# B&R Automation Studio project simulation_of_controlling_the_barn_door
Automation Studio 4.2.10.53 SP

## Configuration SampleText

CPU 4PP065.0571-P74, AutomationRuntime D4.26, Build 4.1.2, Vc V4.25.0, Safety 1.6

### Task classes (Cpu.sw)
```
Cyclic#1 (cycle 2000 us, tolerance 0 us):
  ncsdcctrl <- ncsdcctrl.prg
Cyclic#4 (cycle 100000 us, tolerance 100000 us):
  Program <- Program.prg
NcDataObjects: acp10etxen <- acp10etxen.dob, gAxis01a <- gAxis01obj.gAxis01a.dob, gAxis01i <- gAxis01obj.gAxis01i.dob
Libraries: Acp10sdc, sys_lib, Runtime, asstring, Acp10man, Acp10par, NcGlobal, Acp10_MC, brsystem, AsBrStr, Library
```

### Hardware
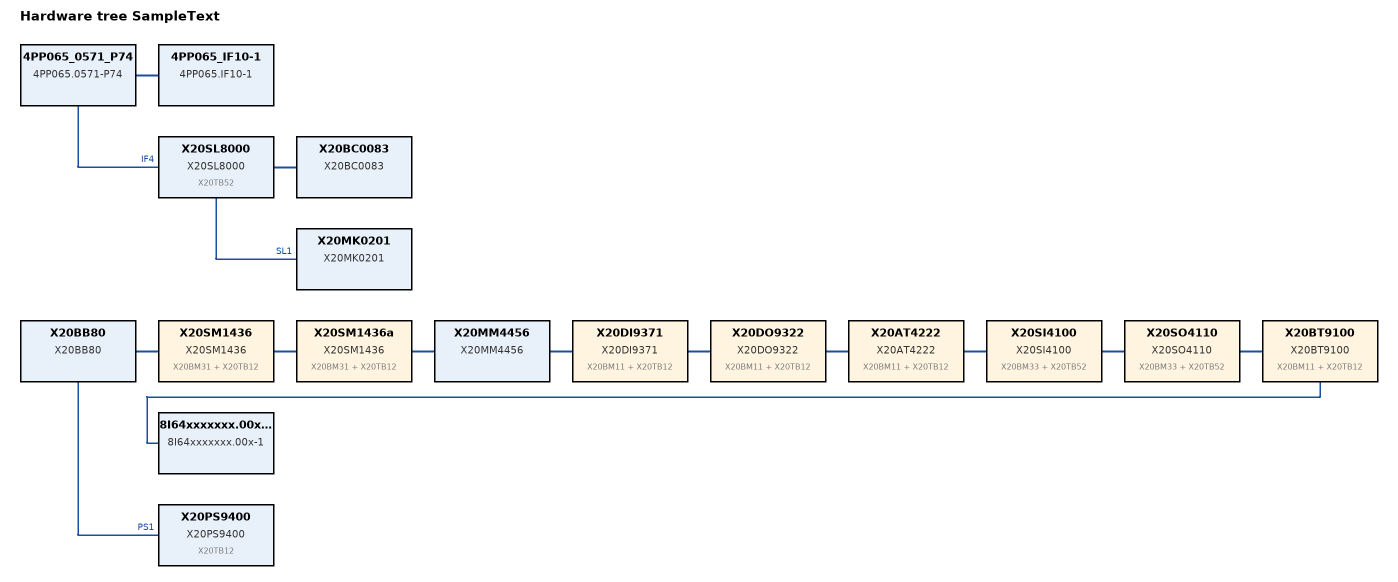
```
4PP065_0571_P74 : 4PP065.0571-P74 v1.1.1.0
  Connector IF4:
    EplInterfaceRedundant = 0
    EplEthInterfaceRedundant = 0
  Connector IF5:
    ActivateDevice = 1
    Mode = Manual
    InternetAddress = 10.1.1.13
    SubnetMask = 255.255.255.0
  ConfigurationID = DriveControl_SampleText
  TimerDeviceType = EPLX2X
  TimerDevice = 4PP065_0571_P74.IF4
  TaskClassIdleTime = 2000
  Cyclic1Duration = 2000
  Cyclic1Tolerance = 0
  Cyclic1Output = 1
  Cyclic2Duration = 20000
  Cyclic2Tolerance = 20000
  Cyclic3Duration = 50000
  Cyclic3Tolerance = 50000
  Cyclic4Duration = 100000
  Cyclic4Tolerance = 100000
  Cyclic5Duration = 200000
  Cyclic5Tolerance = 200000
  Cyclic6Duration = 500000
  Cyclic6Tolerance = 500000
  Cyclic7Duration = 1000000
  Cyclic7Tolerance = 1000000
  Cyclic8Duration = 10000
  Cyclic8Tolerance = 30000000
4PP065_IF10-1 : 4PP065.IF10-1 v1.0.2.0  [SS -> 4PP065_0571_P74.SS1]
8I64xxxxxxx.00x-1 : 8I64xxxxxxx.00x-1 v1.3.8.5  [X2X1 -> X20BT9100.X2X1]
  packedETAD = packed
  packedETI = packed
  packedCMDD = packed
  packedCMI = packed
  ACC = 30
X20AT4222 : X20AT4222 v1.2.1.0  [SS1 -> X20TB12e.SS; SL -> X20BM11c.SL1]
X20BB80 : X20BB80 v1.0.0.2
X20BC0083 : X20BC0083 v2.5.0.0  [PLK1 -> X20SL8000.PLK2 (NodeNumber=2); SL -> X20BB80.SL1]
X20BM11 : X20BM11 v1.0.0.1  [X2X1 -> X20BM33a.X2X2]
X20BM11a : X20BM11 v1.0.0.1  [X2X1 -> X20MM4456.X2X2]
X20BM11b : X20BM11 v1.0.0.1  [X2X1 -> X20BM11a.X2X2]
X20BM11c : X20BM11 v1.0.0.1  [X2X1 -> X20BM11b.X2X2]
X20BM31 : X20BM31 v1.0.0.1  [X2X1 -> X20BB80.IF1]
X20BM31a : X20BM31 v1.0.0.1  [X2X1 -> X20BM31.X2X2]
X20BM33 : X20BM33 v1.0.0.4  [X2X1 -> X20BM11c.X2X2]
X20BM33a : X20BM33 v1.0.0.4  [X2X1 -> X20BM33.X2X2]
X20BT9100 : X20BT9100 v1.0.2.4  [SS1 -> X20TB12f.SS; SL -> X20BM11.SL1]
X20DI9371 : X20DI9371 v1.0.1.3  [SS1 -> X20TB12c.SS; SL -> X20BM11a.SL1]
X20DO9322 : X20DO9322 v1.0.3.0  [SS1 -> X20TB12d.SS; SL -> X20BM11b.SL1]
X20MK0201 : X20MK0201 v1.0.0.0  [SL -> X20SL8000.SL1]
X20MM4456 : X20MM4456 v1.1.3.1  [X2X1 -> X20BM31a.X2X2]
X20PS9400 : X20PS9400 v1.0.2.4  [SS1 -> X20TB12.SS; PS -> X20BB80.PS1]
X20SI4100 : X20SI4100 v1.10.0.1  [SS1 -> X20TB52.SS; SL -> X20BM33.SL1]
X20SL8000 : X20SL8000 v1.6.5.1  [PLK1 -> 4PP065_0571_P74.IF4 (NodeNumber=1); PLK2 -> X20BC0083.PLK1 (NodeNumber=1); SS1 -> X20TB52b.SS]
  SafeProject = SafeLOGIC-1
X20SM1436 : X20SM1436 v1.4.2.0  [SS1 -> X20TB12a.SS; SL -> X20BM31.SL1]
X20SM1436a : X20SM1436 v1.4.2.0  [SS1 -> X20TB12b.SS; SL -> X20BM31a.SL1]
X20SO4110 : X20SO4110 v1.10.0.1  [SS1 -> X20TB52a.SS; SL -> X20BM33a.SL1]
  SafeModuleID = 3
X20TB12 : X20TB12 v1.0.0.0
X20TB12a : X20TB12 v1.0.0.0
X20TB12b : X20TB12 v1.0.0.0
X20TB12c : X20TB12 v1.0.0.0
X20TB12d : X20TB12 v1.0.0.0
X20TB12e : X20TB12 v1.0.0.0
X20TB12f : X20TB12 v1.0.0.0
X20TB52 : X20TB52 v1.0.0.1
X20TB52a : X20TB52 v1.0.0.1
X20TB52b : X20TB52 v1.0.0.1
```

### IoMap.iom - 4PP065_0571_P74/IoMap.iom
```iecst
VAR_CONFIG
	Cyclic#1.gAxis01_DrvIf.iLifeCnt AT %IB."8I64xxxxxxx.00x-1".SDC_LifeCnt;
	Cyclic#1.gAxis01_DrvIf.oSetTime AT %QW."8I64xxxxxxx.00x-1".SDC_SetTime;
	Cyclic#1.gAxis01_DrvIf.oSetPos AT %QW."8I64xxxxxxx.00x-1".LFRD_Output;
	Cyclic#1.gAxis01_DiDoIf.iLifeCntDriveReady AT %IB."8I64xxxxxxx.00x-1".SDC_LifeCnt;
	Cyclic#1.gAxis01_DiDoIf.iLifeCntDriveEnable AT %IB."8I64xxxxxxx.00x-1".SDC_LifeCnt;
	Cyclic#1.gAxis01_ModuleOk AT %IX."8I64xxxxxxx.00x-1".ModuleOk;
	::Program:FBDoorSM.direction AT %IX."X20DI9371".DigitalInput01;
	::Program:FBDoorSM.sw1 AT %IX."X20DI9371".DigitalInput02;
	::Program:FBDoorSM.sw2 AT %IX."X20DI9371".DigitalInput03;
	::Program:FBDoorSM.sw3 AT %IX."X20DI9371".DigitalInput04;
	::Program:FBDoorSM.sw4 AT %IX."X20DI9371".DigitalInput05;
	::Program:FBLedSM.led1 AT %QX."X20DO9322".DigitalOutput01;
	::Program:FBLedSM.led2 AT %QX."X20DO9322".DigitalOutput02;
	::Program:FBLedSM.led3 AT %QX."X20DO9322".DigitalOutput03;
	::Program:FBLedSM.led4 AT %QX."X20DO9322".DigitalOutput04;
	::Program:FBDriveSM.state AT %IW."8I64xxxxxxx.00x-1".ETAD_Input;
	::Program:FBDriveSM.command AT %IW."8I64xxxxxxx.00x-1".ETI_Input;
	::Program:FBDriveSM.speed AT %IW."8I64xxxxxxx.00x-1".RFRD_Input;
END_VAR
```

## Logical view

Binary libraries used (declarations not repeated): Runtime, Operator, AsIecCon, astime, sys_lib, asstring, Acp10sdc 3.16.2, Acp10man 3.16.2, Acp10par 3.16.2, NcGlobal 3.16.2, Acp10_MC 3.16.2, brsystem, AsBrStr


### Program Logical/ncsdcctrl (IEC)

#### ncsdcctrlInit.st
```iecst
PROGRAM _INIT

(* ### BEGIN gAxis01 ### *)

(* initialize variables *)
        gAxis01_HW.DrvIf_Typ := ncSDC_DRVSERVO16;
        brsstrcpy( ADR(gAxis01_HW.DrvIf_Name[0]), ADR('gAxis01_DrvIf') );
        gAxis01_HW.DiDoIf_Typ := ncSDC_DIDO;
        brsstrcpy( ADR(gAxis01_HW.DiDoIf_Name[0]), ADR('gAxis01_DiDoIf') );

(* force variable offset generation *)
        gAxis01.size                      := gAxis01.size;
        gAxis01_DrvIf.iLifeCnt            := gAxis01_DrvIf.iLifeCnt;
        gAxis01_DiDoIf.iLifeCntDriveReady := gAxis01_DiDoIf.iLifeCntDriveReady;
        gAxis01_ModuleOk                  := gAxis01_ModuleOk;

(* assign your hardware inputs here*)

(*      gAxis01_DiDoIf.iPosHwEnd  := gAxis01_DiDoIf.iPosHwEnd;
        gAxis01_DiDoIf.iNegHwEnd  := gAxis01_DiDoIf.iNegHwEnd;
        gAxis01_DiDoIf.iReference := gAxis01_DiDoIf.iReference;
 *)

(* ### END gAxis01 ### *)

END_PROGRAM
```

### Library Logical/Library (ANSIC)

#### Types.typ - Exported data types
```iecst
TYPE
	DoorSM :
		(
		ST_INIT,
		ST_UNKNOWN,
		ST_OPEN,
		ST_CLOSE,
		ST_ACC_POS,
		ST_ACC_NEG,
		ST_POS,
		ST_NEG,
		ST_DEC_POS,
		ST_DEC_NEG
		);
	StateOfFreqConv :
		(
		DISABLED,
		SWITCHED_ON,
		READY
		);
	CommandToDoor :
		(
		CMD_SWITCH_ON,
		CMD_SHUTDOWN,
		CMD_ENABLE
		);
END_TYPE
```

#### Library.fun - Exported functions and function blocks
```iecst
FUNCTION_BLOCK FB_LedSM (*TODO: Add your comment here*) (*$GROUP=User,$CAT=User,$GROUPICON=User.png,$CATICON=User.png*)
	VAR_INPUT
		state : UINT;
	END_VAR
	VAR_OUTPUT
		led1 : BOOL;
		led2 : BOOL;
		led3 : BOOL;
		led4 : BOOL;
		timer : INT;
	END_VAR
END_FUNCTION_BLOCK

FUNCTION_BLOCK FB_DoorSM (*TODO: Add your comment here*) (*$GROUP=User,$CAT=User,$GROUPICON=User.png,$CATICON=User.png*)
	VAR_INPUT
		state : UINT;
		sw1 : BOOL;
		sw2 : BOOL;
		sw3 : BOOL;
		sw4 : BOOL;
		direction : BOOL;
	END_VAR
	VAR_OUTPUT
		speed : INT;
	END_VAR
END_FUNCTION_BLOCK

FUNCTION_BLOCK FB_DriveSM (*TODO: Add your comment here*) (*$GROUP=User,$CAT=User,$GROUPICON=User.png,$CATICON=User.png*)
	VAR_INPUT
		state : UINT;
		enable : BOOL;
	END_VAR
	VAR_OUTPUT
		command : UINT;
		speed : INT;
	END_VAR
END_FUNCTION_BLOCK
```

#### FB_LedSM.c
```c
#include <bur/plctypes.h>
#ifdef __cplusplus
	extern "C"
	{
#endif
	#include "Library.h"
#ifdef __cplusplus
	};
#endif
/* TODO: Add your comment here */
void FB_LedSM(struct FB_LedSM* inst)
{
	switch(inst->state)
	{
		case ST_INIT:
			{
				break;
			}
		case ST_UNKNOWN:
			{
				if(inst->timer%10 == 9)
				{
					inst->led0 = !inst->led0;
					inst->led1 = !inst->led1;
					inst->led2 = !inst->led2;
					inst->led3 = !inst->led3;
				}
				break;
			}
		case ST_OPEN:
			{
				inst->led0 = 0;
				inst->led1 = 0;
				inst->led2 = 0;
				inst->led3 = 0;
				break;
			}
		case ST_CLOSE:
			{
				inst->led0 = 1;
				inst->led1 = 1;
				inst->led2 = 1;
				inst->led3 = 1;
				break;
			}
		case ST_ACC_POS:
			{
				if(inst->timer%10 == 4) inst->led0 = 1;
				inst->led1 = 0;
				inst->led2 = 0;
				inst->led3 = 0;
				break;
			}
		case ST_ACC_NEG:
			{
				inst->led0 = 1;
				inst->led1 = 1;
				inst->led2 = 1;
				if(inst->timer%10 == 4) inst->led3 = 0;
				break;
			}
		case ST_POS:
			{
				inst->led0 = 1;
				if(inst->timer%10 == 9) inst->led1 = 1;
				inst->led2 = 0;
				inst->led3 = 0;
				break;
			}
		case ST_NEG:
			{
				inst->led0 = 1;
				inst->led1 = 1;
				if(inst->timer%10 == 9) inst->led2 = 0;
				inst->led3 = 0;
				break;
			}
		case ST_DEC_POS:
			{
				inst->led0 = 1;
				inst->led1 = 1;
				if(inst->timer%10 == 4) inst->led2 = 1;
				inst->led3 = 0;
				break;
			}
		case ST_DEC_NEG:
			{
				inst->led0 = 1;
				if(inst->timer%10 == 4) inst->led1 = 0;
				inst->led2 = 0;
				inst->led3 = 0;
				break;
			}
	}
}
```

#### FB_DoorSM.c
```c
#include <bur/plctypes.h>
#ifdef __cplusplus
	extern "C"
	{
#endif
	#include "Library.h"
#ifdef __cplusplus
	};
#endif
/* TODO: Add your comment here */
void FB_DoorSM(struct FB_DoorSM* inst)
{
	switch(inst->state)
	{
		case ST_INIT:
			{
				if(inst->sw0 == 0 && inst->sw1 == 0 && inst->sw2 == 0 && inst->sw3 == 0) inst->state = ST_UNKNOWN;
				break;
			}
		case ST_UNKNOWN:
			{
				if(inst->direction == 0 && inst->sw0 == 0) inst->state = ST_OPEN;
				if(inst->direction == 1 && inst->sw3 == 1) inst->state = ST_CLOSE;
				break;
			}
		case ST_OPEN:
			{
				inst->speed = 0;
				if(inst->direction == 0) inst->state = ST_ACC_POS;
				break;
			}
		case ST_CLOSE:
			{
				inst->speed = 0;
				if(inst->direction == 1) inst->state = ST_ACC_NEG;
				break;
			}
		case ST_ACC_POS:
			{
				inst->speed = 25;
				if(inst->sw1 == 1) inst->state = ST_POS;
				if(inst->direction == 1) inst->state = ST_DEC_NEG;
				break;
			}
		case ST_ACC_NEG:
			{
				inst->speed = -25;
				if(inst->sw2 == 0) inst->state = ST_NEG;
				if(inst->direction == 0) inst->state = ST_DEC_POS;
				break;
			}
		case ST_POS:
			{
				inst->speed = 5;
				if(inst->sw2 == 1) inst->state = ST_DEC_POS;
				if(inst->direction == 1) inst->state = ST_NEG;
				break;
			}
		case ST_NEG:
			{
				inst->speed = -5;
				if(inst->sw2 == 0) inst->state = ST_DEC_NEG;
				if(inst->direction == 0) inst->state = ST_POS;
				break;
			}
		case ST_DEC_POS:
			{
				inst->speed = 5;
				if(inst->sw3 == 1) inst->state = ST_CLOSE;
				break;
			}
		case ST_DEC_NEG:
			{
				inst->speed = -5;
				if(inst->sw3 == 0) inst->state = ST_OPEN;
				break;
			}
}
```

#### FB_DriveSM.c
```c
#include <bur/plctypes.h>
#ifdef __cplusplus
	extern "C"
	{
#endif
	#include "Library.h"
#ifdef __cplusplus
	};
#endif
/* TODO: Add your comment here */
void FB_DriveSM(struct FB_DriveSM* inst)
{
	if(inst->enable == 1)
	{
		switch(inst->state & 0x6F)
		{
			case ST_DISABLE:
				inst->command = CMD_SHUTDOWN;
				break;
			case ST_SWITCHED_ON:
				inst->command = CMD_SWITCH_ON;
				break;
			case ST_READY:
				inst->command = CMD_ENABLE;
				break;
		}
	}
	else inst->command = CMD_SHUTDOWN;
}
```

### Program Logical/Program (ANSIC)

#### Variables.var
```iecst
VAR
	FBDoorSM : FB_DoorSM := (0);
	FBLedSM : FB_LedSM := (0);
	FBDriveSM : FB_DriveSM := (0);
END_VAR
```

#### Main.c
```c
#include <bur/plctypes.h>

#ifdef _DEFAULT_INCLUDES
	#include <AsDefault.h>
#endif

void _INIT ProgramInit(void)
{
	FBDriveSM.enable = 1;
}

void _CYCLIC ProgramCyclic(void)
{
	FB_DoorSM(&FBDoorSM);

	FBDriveSM.speed = FBDoorSM.speed;
	FB_DriveSM(&FBDriveSM);

	FBLedSM.state = FBDoorSM.state;
	FB_LedSM(&FBLedSM);
	FBLedSM.timer++;

}

void _EXIT ProgramExit(void)
{
	// Insert code here

}
```

Listed in the project but not available here: Logical/Global.typ, Logical/Global.var, Logical/ncsdcctrl/ncsdcctrlCyclic.st, Logical/ncsdcctrl/ncsdcctrl.typ, Logical/ncsdcctrl/ncsdcctrl.var, Logical/acp10etxen, Logical/gAxis01obj, Logical/Library/Constants.var
